PROGRAM P_FeedForward
VAR
	fbFF : FB_FeedForward;
END_VAR

fbFF(
	fMaxFlowUp := G_Parameter.fQMaxUp,
	fMaxFlowDown := G_Parameter.fQMaxDown,
	fDeadUp := G_Parameter.fDeadUp,
	fDeadDown := G_Parameter.fDeadDown,
	fAreaUp := G_Parameter.fAreaUp,
	fAreaDown := G_Parameter.fAreaDown,
	
	fPs := G_OPC.fPs,
	fPa := G_OPC.fPa,
	fPb := G_OPC.fPb,
	fDeltaP0 := G_Parameter.fDeltaP0,
);

IF TO_BOOL(G_Inputs.bAuto) THEN
	fbFF(
		fXDotRef := G_OPC.fXDotRef,		
		
		fUFF => G_OPC.fFF,
	);


ELSIF TO_BOOL(G_Inputs.bManual) THEN
	fbFF(
		fXDotRef := G_OPC.fJoystick * G_Parameter.fMaxSpeed,
		
		fUFF => G_OPC.fFF,
	);

END_IF

END_PROGRAM

(* stored: Version 1.1.0.1, ProductVersion 3.1.4024.12
   POU P_FeedForward: Id {202d862f-f86c-42e9-b9cf-42d47a621534}, SpecialFunc None *)
